FUNCTION_BLOCK PumpControl
VAR_INPUT
	ManAutoPb			:	BOOL;			// Manual / auto mode; TRUE=Manual
	ManPumpStart		:	BOOL;			// Command Pump On in Manual Mode (N.O.)
	ManPumpStop			:	BOOL;			// Command Pump Off in Manual Mode (N.C)
	LevelSensorMin		:	BOOL;			// Tank low level sensor (N.C)
	LevelSensorMax		:	BOOL;			// Tank high level sensor (N.C)
END_VAR
VAR_OUTPUT
	PumpRunning			:	BOOL;			// Motor pump RUN state
	ManAutoState		:	BOOL;			// Indication of manual / auto mode
END_VAR
VAR
	srPumpRunning		: SR;
	PumpOffCommand		: BOOL;
	tonDelay			: TON;
	rtrigManAuto		: R_TRIG;
END_VAR

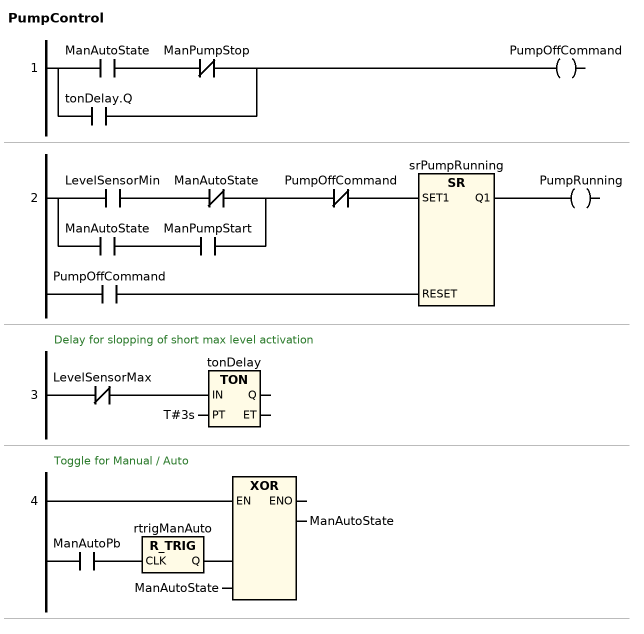
// NETWORK 1
PumpOffCommand := ManAutoState AND NOT ManPumpStop OR tonDelay.Q;

// NETWORK 2
srPumpRunning(SET1 := (LevelSensorMin AND NOT ManAutoState OR ManAutoState AND ManPumpStart) AND NOT PumpOffCommand, RESET := PumpOffCommand); // SR
PumpRunning := srPumpRunning.Q1;

// NETWORK 3
// Delay for slopping of short max level activation
tonDelay(IN := NOT LevelSensorMax, PT := T#3s); // TON

// NETWORK 4
// Toggle for Manual / Auto
rtrigManAuto(CLK := ManAutoPb); // R_TRIG
ManAutoState := rtrigManAuto.Q XOR ManAutoState;

END_FUNCTION_BLOCK

(* stored: Version 1.1.0.1, ProductVersion 3.1.4024.15
   POU PumpControl: Id {f1099f5a-b944-4061-a6b4-9e970b277656}, SpecialFunc None *)
